FUNCTION_BLOCK IO_WRITER
  (* Standard: 61499-2 *)
  (* Version 11-01-12, IECVM *)
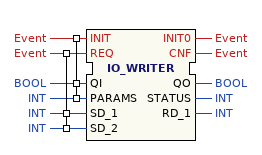
  EVENT_INPUT
    INIT WITH QI, PARAMS;
    REQ WITH SD_1, SD_2;
  END_EVENT
  EVENT_OUTPUT
    INIT0;
    CNF;
  END_EVENT
  VAR_INPUT
    QI : BOOL;
    PARAMS : INT;
    SD_1 : INT;
    SD_2 : INT;
  END_VAR
  VAR_OUTPUT
    QO : BOOL;
    STATUS : INT;
    RD_1 : INT;
  END_VAR
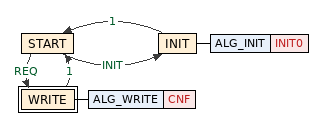
  EC_STATES
    WRITE : ALG_WRITE -> CNF;
    START;
    INIT : ALG_INIT -> INIT0;
  END_STATES
  EC_TRANSITIONS
    START TO INIT := INIT;
    INIT TO START := 1;
    START TO WRITE := REQ;
    WRITE TO START := 1;
  END_TRANSITIONS
  ALGORITHM ALG_WRITE IN Lua:
SET_REG(SD_1, SD_2);
  END_ALGORITHM
  ALGORITHM ALG_INIT IN Lua:

  END_ALGORITHM
END_FUNCTION_BLOCK
